// Mitsubishi GX Works2 project: 241010_금석통과비금석배출   PLC: Q03UDV

PROGRAM MAIN
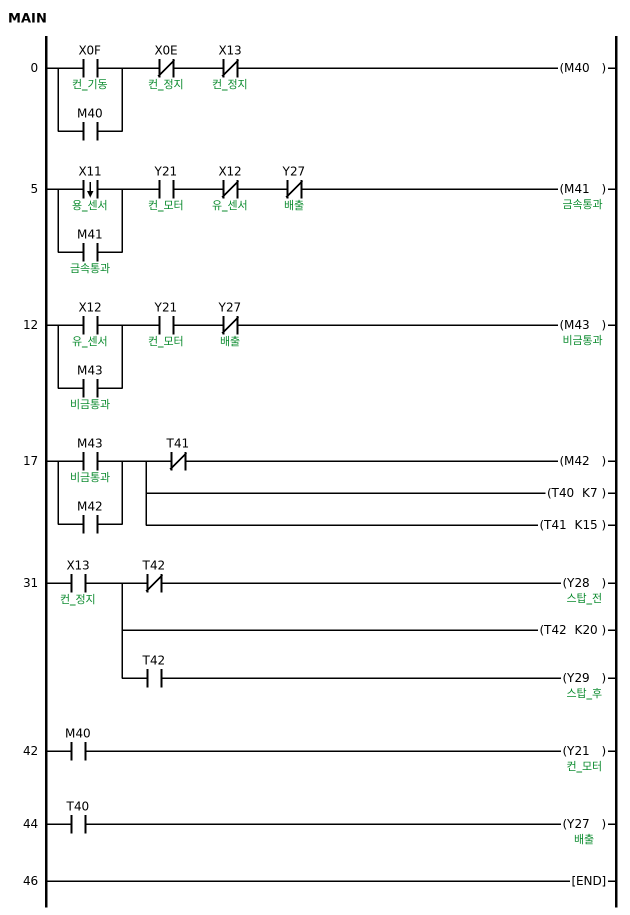
0     LD      X0F  ; 컨_기동
      OR      M40
      ANI     X0E  ; 컨_정지
      ANI     X13  ; 컨_정지
      OUT     M40
5     LDF     X11  ; 용_센서
      OR      M41  ; 금속통과
      AND     Y21  ; 컨_모터
      ANI     X12  ; 유_센서
      ANI     Y27  ; 배출
      OUT     M41  ; 금속통과
12    LD      X12  ; 유_센서
      OR      M43  ; 비금통과
      AND     Y21  ; 컨_모터
      ANI     Y27  ; 배출
      OUT     M43  ; 비금통과
17    LD      M43  ; 비금통과
      OR      M42
      MPS
      ANI     T41
      OUT     M42
      MPP
      OUT     T40 K7
      OUT     T41 K15
31    LD      X13  ; 컨_정지
      MPS
      ANI     T42
      OUT     Y28  ; 스탑_전
      MPP
      OUT     T42 K20
      AND     T42
      OUT     Y29  ; 스탑_후
42    LD      M40
      OUT     Y21  ; 컨_모터
44    LD      T40
      OUT     Y27  ; 배출
46    END
END_PROGRAM
